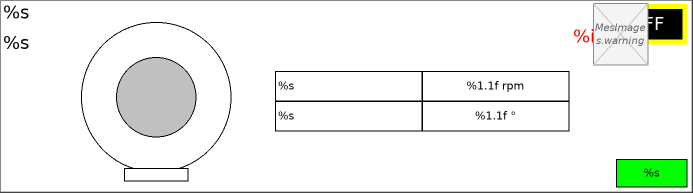
VISUALIZATION VISU_AXE_STD1_ROT_ABS_FCT_ETAT_OSC  // 693x193
VAR_IN_OUT
	m_Input_MOTEUR: BLOCK_AXE_STD1_OSCILLANT;
	m_Input_PRG_MOUVEMENT_PS: BLOCK_PRG_MOUVEMENT_PS;
END_VAR
VAR_INPUT CONSTANT
	m_Input_ID_NOM_XML : INT;
	m_Input_INDEX_MOTEUR : INT;
END_VAR
    Rectangle (0,0 693x193), "%s", text list: 'TextList_Type_Moteur', text index: m_Input_ID_NOM_XML
    Rectangle (0,28 107x30), "%s", text variable: m_Input_MOTEUR.MNEMO
    RoundedRectangle (275,71 147x30), "%s", text list: 'TextList_Moteurs', text index: 7
    RoundedRectangle (275,101 147x30), "%s", text list: 'TextList_Moteurs', text index: 12
    RoundedRectangle (422,71 147x30), "%1.1f rpm", text variable: m_Input_MOTEUR.STATE_Vit
    RoundedRectangle (422,101 147x30), "%1.1f °", text variable: m_Input_MOTEUR.STATE_Pos
    Group (81,22 150x150), invisible if: NOT m_Input_PRG_MOUVEMENT_PS.CONF_Poste_Central[m_Input_INDEX_MOTEUR]
        Ellipse (0,0 150x150)
        Ellipse (35,35 80x80)
    Rectangle (124,168 64x13)
    RoundedRectangle (607,4 80x40), invisible if: NOT m_Input_MOTEUR.OP_Validation.OK
    RoundedRectangle (607,4 80x40), invisible if: NOT m_Input_MOTEUR.OP_Validation.AR
    RoundedRectangle (607,4 80x40), invisible if: NOT m_Input_MOTEUR.OP_Validation.EC
    RoundedRectangle (612,9 70x30), "ON", invisible if: m_Input_MOTEUR.STATE_Ar
    RoundedRectangle (612,9 70x30), "OFF", invisible if: NOT m_Input_MOTEUR.STATE_Ar
    Rectangle (531,24 67x21), "%i", text variable: m_Input_MOTEUR.STATE_Err, invisible if: NOT m_Input_MOTEUR.STATE_NOK
    Image (593,3 55x62), invisible if: NOT m_Input_MOTEUR.STATE_NOK, image: MesImages.warning
    RoundedRectangle (616,159 71x28), "%s", invisible if: m_Input_MOTEUR.STATE_Homed OR m_Input_MOTEUR.CONF_No_Ref, text list: 'TextList_Moteurs', text index: 11
    RoundedRectangle (616,159 71x28), "%s", invisible if: NOT m_Input_MOTEUR.STATE_Homed OR m_Input_MOTEUR.CONF_No_Ref, text list: 'TextList_Moteurs', text index: 11
END_VISUALIZATION

(* stored: Version 1.1.0.1, ProductVersion 3.1.4024.10
   Visu VISU_AXE_STD1_ROT_ABS_FCT_ETAT_OSC: Id {bc471759-9d23-4570-9960-d6643d6b57e5} *)
